TYPE EM_Filling_HMI :
STRUCT
	Start		: BOOL;
	Stop		: BOOL;
	Reset		: BOOL;
	Abort		: BOOL;
	Richting_L	: BOOL;
	Richting_R	: BOOL;
	Toerental	: INT;
	Auto		: BOOL;
	Manueel		: BOOL;
	Clear		: BOOL;
	UnSuspend	: BOOL;
	Suspend		: BOOL;
	UnHold		: BOOL;
	Hold		: BOOL;
END_STRUCT
END_TYPE

(* stored: Version 1.1.0.1, ProductVersion 3.1.4024.12
   DUT EM_Filling_HMI: Id {61fd04d5-eccf-4b2e-98b4-ca35c6dc47ed} *)
